	        // Buttons control
	        // Mains
	        IF (#statAvailAct3Mains = FALSE) THEN
	            #statAction.start := FALSE;
	            #statAction.stop := FALSE;
	            #statAction.end := FALSE;
	            
	        END_IF;
	        
	        // Cancel
	        IF (#statAvailActCancel = FALSE) THEN
	            #statAction.cancel := FALSE;
	            
	        END_IF;
	        
	        // Confirm
	        IF (#statAvailActConfirm = FALSE) THEN
	            #statAction.confirm := FALSE;
	            
	        END_IF;
	        
	        // Reset time
	        IF (#statAvailActResetTime = FALSE) THEN
	            #statAction.resetTime := FALSE;
	            
	        END_IF;
	        
	        // Action: Collective integer
	        "AFC_Struct_To_Word"(s := #statAction,
	                             w => #tempAction);
	        
	        #action := WORD_TO_INT(#tempAction);
	        
	    END_REGION reset availability and latching buttons
	    
	END_REGION CONTROL OPTIONS
	
	REGION WRITE OUTPUTS
	    // Outputs
	    #availAct3Mains := #statAvailAct3Mains;
	    #availActCancel := #statAvailActCancel;
	    #availActConfirm := #statAvailActConfirm;
	    #availActResetTime := #statAvailActResetTime;
	    
	END_REGION WRITE OUTPUTS
END_FUNCTION_BLOCK

FUNCTION_BLOCK "AFB_Sequencer"
TITLE = AFB_Sequencer1
{ S7_Optimized_Access := 'TRUE' }
AUTHOR : CH
FAMILY : Aktina
NAME : SEQUENCER
VERSION : 0.1
//AFB_Sequencer1
   VAR_INPUT 
      p1s : Bool;   //  TRUE: 1 pulse every 1s
      startAllow : Bool;   //  TRUE: The sequencer start condition is valid and it is allowed to start
      startCond : Bool;   //  TRUE: The options controller released the condition for the booting of the sequencer
      endCond : Bool;   //  TRUE: The state machine should end its execution immediately
      runcond : Bool;   //  TRUE: The option is running
      resetTimeOut : Bool;   //  TRUE: The time out timer should reset
      offset : Int;   //  Offset number for active step
      holdReset : DInt;   //  Preset time after the end of the sequencer to block restarting
      stepSP : Array[0..#ctMAX_STEP] of "dtStepSP";   //  Array containing the steps setpoints
      stepCond : Array[0..#ctMAX_STEP] of "dtStepCond";   //  Array containing all the steps conditions
   END_VAR

   VAR_OUTPUT 
      blocked : Bool;   //  TRUE: The sequencer is blocked from starting
      timeout : Bool;   //  TRUE: The sequencer execution has timed out
      busy : Bool;   //  TRUE: The sequencer has started and it is ongoing
      run : Bool;   //  TRUE: The sequencer operation is running
      prompt : Bool;   //  TRUE: The sequencer prompts for an operator confirmation
      error : Bool;   //  TRUE: An error was generated during execution
      noFault : Bool;   //  TRUE: The active step is running without errors
      done : Bool;   //  TRUE: The sequencer execution has finished
      terminate : Bool;   //  TRUE: The sequencer execution was terminated either by force of error
      fin : Bool;   //  TRUE: The sequencer end timer has just expired (stays high for 1 cycle)
      stepOn : Array[0..#ctMAX_STEP] of Bool;   //  TRUE: The step has just been loaded
      stepAct : Array[0..#ctMAX_STEP] of Bool;   //  TRUE: The step is active
      stepRun : Array[0..#ctMAX_STEP] of Bool;   //  TRUE: The step is running (used mostly as condition for activations)
      stepOff : Array[0..#ctMAX_STEP] of Bool;   //  TRUE: The step has just ended
      status : Word;   //  Status of the function block
      stepNr : Int;   //  Number of active step = offset + statFBState
      stateNr : Int;   //  Number of active state = statFBState
   END_VAR

   VAR RETAIN
      statStartReqOld { ExternalAccessible := 'False'; ExternalVisible := 'False'; ExternalWritable := 'False'} : Bool;
      statFBState { ExternalWritable := 'False'} : Int := #ctFB_STATE_NO_PROCESSING;   //  State in the state machine of the FB
      statStatus { ExternalWritable := 'False'} : Word := #ctSTATUS_NO_CALL;   //  Static value for output 'status'
   END_VAR
   VAR DB_SPECIFIC
      statBusy { ExternalAccessible := 'False'; ExternalVisible := 'False'; ExternalWritable := 'False'} : Bool;   //  Static value for output 'busy'
      statRun { ExternalAccessible := 'False'; ExternalVisible := 'False'; ExternalWritable := 'False'} : Bool;   //  Static value for output 'run'
      statPrompt { ExternalAccessible := 'False'; ExternalVisible := 'False'; ExternalWritable := 'False'} : Bool;   //  Static value for output 'prompt'
      statError { ExternalAccessible := 'False'; ExternalVisible := 'False'; ExternalWritable := 'False'} : Bool;   //  Static value for output 'error'
      statNoFault { ExternalAccessible := 'False'; ExternalVisible := 'False'; ExternalWritable := 'False'} : Bool;   //  Static value for output 'noFault'
      statDone { ExternalAccessible := 'False'; ExternalVisible := 'False'; ExternalWritable := 'False'} : Bool;   //  Static value for output 'done'
      statTerminate { ExternalAccessible := 'False'; ExternalVisible := 'False'; ExternalWritable := 'False'} : Bool;   //  Static value for output 'terminate'
      statFin { ExternalAccessible := 'False'; ExternalVisible := 'False'; ExternalWritable := 'False'} : Bool;   //  Static value for output 'fin'
      statExclude { S7_SetPoint := 'True'} : Bool;   //  Static value that allows the supervisor to stop the forced step updating from the current step
      statForce { S7_SetPoint := 'True'} : Bool;   //  Static value that allows the supervisor to force a new step
      statLastStep : Int;   //  Static value for the last step number
      statForceStep { S7_SetPoint := 'True'} : Int;   //  Static value for the new forced step value
   END_VAR
   VAR 
      statStepOn : Array[0..#ctMAX_STEP] of Bool;   //  Static memory area for output array "stepOn"
      statStepAct : Array[0..#ctMAX_STEP] of Bool;   //  Static memory area for output array "stepOn"
      statStepRun : Array[0..#ctMAX_STEP] of Bool;   //  Static memory area for output array "stepRun"
      statStepOff : Array[0..#ctMAX_STEP] of Bool;   //  Static memory area for output array "stepOff"
   END_VAR
   VAR RETAIN
      instTimeReset {InstructionName := 'IEC_TIMER'; LibVersion := '1.0'; S7_SetPoint := 'False'} : IEC_TIMER;   //  Instance for the timer that resets everything and prevents restarting
   END_VAR
   VAR 
      instTimeStep { S7_SetPoint := 'False'} : "AFB_TimeCount";   //  Instance for the step timer
      instTimeOut { S7_SetPoint := 'False'} : "AFB_TimeCount";   //  Instance for the timeout timer
   END_VAR

   VAR_TEMP 
      tempStartAllow : Bool;   //  Temporary status bit for the "startAllow" input
      tempStartCond : Bool;   //  Temporary status bit for the "startCond" input
      tempEndCond : Bool;   //  Temporary status bit for the "endCond" input
      tempRun : Bool;   //  Temporary status bit for the "run" input
      tempChangeStep : Bool;   //  Temporary status bit set whenever a change of step is required
      tempForceStep : Bool;   //  Temporary status bit set whenever a forcing of step is required
      tempStepSP : "dtStepSP";   //  Temporary area for the active step setpoints
      tempStepCond : "dtStepCond";   //  Temporary area for the active step conditions
      n : Int;   //  Temporary LOOP operand
   END_VAR

   VAR CONSTANT 
      ctMAX_STEP : Int := 31;   //  Max: Number steps
      ctMAX_HOPS : Int := 31;   //  Max: Hops allowed for the while loop
      ctFB_STATE_NO_PROCESSING : Int := 0;   //  FB state: No processing
      ctFB_STATE_PROCESSING_1 : Int := 1;   //  FB state: Processing 1
      ctSTATUS_NO_CALL : Word := 16#7000;   //  Status: No job being currently processed
      ctSTATUS_FIRST_CALL : Word := 16#7001;   //  Status: First call after incoming new job (rising edge 'execute')
      ctSTATUS_SUBSEQUENT_CALL : Word := 16#7002;   //  Status: Subsequent call during active processing without further details
      ctSTATUS_EXECUTION_TERMINATED : Word := 16#7008;   //  Status: Execution finished without errors
      ctSTATUS_EXECUTION_FINISHED : Word := 16#700F;   //  Status: Execution finished without errors
      ctERR_UNDEFINED_STATE : Word := 16#8000;   //  Error: Due to an undefined state in state machine
      ctERR_IN_BLOCK_OPERATION : Word := 16#8001;   //  Error: Wrong operation of the function block
      ctERR_PARAMETRIZATION : Word := 16#8002;   //  Error: During parameterization
   END_VAR


BEGIN
	REGION BLOCK HEADER
	     //===============================================================================
	     // CH / (c)Copyright (2021)
	     //-------------------------------------------------------------------------------
	     // Title:             (Sequencer control block type 1)
	     // Comment/Function:  (Control step execution of a sequencer by providing only key conditions and setpoints)
	     // Library/Family:    (Aktina/Tools/Sequencer)
	     // Author:            (CH)
	     // Tested with:       (V16)
	     // Engineering:       (TIA Step7 Professional V16)
	     // Restrictions:      ()
	     // Requirements:      (S7-15xx/12xx CPUs)
	     // Notes:             (See block notes)
	     //-------------------------------------------------------------------------------
	     // Change log table:
	     // Version  | Date       | Dev in charge          | Changes
	     //----------|------------|------------------------|------------------------------
	     // 01.00.00 | 2021-08-22 | (CH)                   | First released version
	     // 01.00.01 | 2022-01-13 | (CH)                   | "No timeout" allowed - busy hangon corrected
	     // 01.00.02 | 2023-05-18 | (CH)                   | "RESET(instResetTimer) - removed to allow timer to run
	     //===============================================================================
	END_REGION
	
	REGION BLOCK NOTES
	     //===============================================================================
	     // 1: The number of steps participating is configured by the #ctMAX_STEP
	     //-------------------------------------------------------------------------------
	     // 2: The idle or exit step is always 0 so the number of steps remaining
	     // for the rest of the program is steps = #ctMAX_Step - 1
	     //-------------------------------------------------------------------------------
	     // 3: The block supports zero cycles for step change even if there are 
	     // multiple hops.
	     //-------------------------------------------------------------------------------
	     // 4: The maximum allowed number of hops is the ctMAX_HOPS to avoid an endless
	     // loop. After that alarm is generated.
	     //===============================================================================
	END_REGION
	
	REGION GENERIC PRE-INSTRUCTIONS
	     //  Init temporary area
	     #tempStartAllow := (#startAllow = TRUE) AND (#instTimeReset.Q = FALSE) AND (#statDone = FALSE) AND (#statTerminate = FALSE);
	     #tempStartCond := #startCond;
	     #tempEndCond := #endCond;
	     #tempRun := #runcond;
	     #tempChangeStep := FALSE;
	     #tempForceStep := FALSE;
	     #tempStepSP := #stepSP[0];
	     #tempStepCond := #stepCond[0];
	     #n := 0;
	     
	     // Reset static step memory with every cycle to avoid forced states loaded by a programmer
	     FOR #n := 0 TO #ctMAX_STEP DO
	          #statStepOn[#n] := FALSE;
	          #statStepAct[#n] := FALSE;
	          #statStepRun[#n] := FALSE;
	          #statStepOff[#n] := FALSE;
	     END_FOR;
	     
	END_REGION GENERIC PRE-INSTRUCTIONS
	
	REGION TRIGGERING
	     IF (#tempStartCond = TRUE) AND (#statStartReqOld = FALSE) // Check if FB is triggered
	          AND (#tempStartAllow = TRUE)
	          AND (#tempEndCond = FALSE)
	          AND (#instTimeReset.Q = FALSE)
	          AND (#stepSP[0].next > 0)
	          AND (#statBusy = FALSE)
	          AND (#statDone = FALSE)
	     THEN // First call; initialize FB stat 
	          // TODO: Initialize functionality: reset of variables, diagnostics, etc.
	          #statBusy := TRUE;
	          #statStepOff[0] := TRUE;
	          #statStepAct[0] := FALSE;
	          #statStatus := #ctSTATUS_FIRST_CALL;
	          
	          // TODO: Initialize functionality: start state machine.
	          #statFBState := #stepSP[0].next;
	          
	          // TODO: Initialize functionality: call subsidiary FBs with FALSE
	          "AFC_RESET_TimeCount"(#instTimeStep);
	          "AFC_RESET_TimeCount"(#instTimeOut);
	          RESET_TIMER(#instTimeReset);
	          
	     ELSIF (#statStatus = #ctSTATUS_FIRST_CALL) THEN
	          #statStatus := #ctSTATUS_SUBSEQUENT_CALL;
	     END_IF;
	     
	     // Edge detection 'startReq' input
	     #statStartReqOld := #tempStartCond;
	END_REGION TRIGGERING
	
	REGION END WHEN IDLE
	     IF (#statStatus = #ctSTATUS_NO_CALL) THEN // Nothing to do -> End here to reduce "system load"
	          // Static memory
	          #statDone := FALSE;
	          #statTerminate := FALSE;
	          #statBusy := FALSE;
	          #statRun := FALSE;
	          #statNoFault := TRUE;
	          #statError := FALSE;
	          #statPrompt := FALSE;
	          #statExclude := FALSE;
	          #statForce := FALSE;
	          #statFin := FALSE;
	          #statLastStep := #statFBState;
	          #statForceStep := #statFBState;
	          #statStepAct[0] := TRUE;
	          
	          // if ENO mechanism is not used / not wanted replace the following line by --> ENO := TRUE;
	          // ENO := NOT #statError;
	          ENO := TRUE;
	          
	          // Outputs
	          #blocked := (#startAllow = FALSE);
	          #timeout := FALSE;
	          #done := #statDone;
	          #terminate := #statTerminate;
	          #busy := #statBusy;
	          #run := #statRun;
	          #noFault := #statNoFault;
	          #error := #statError;
	          #prompt := #statPrompt;
	          #fin := #statFin;
	          #stepOn := #statStepOn;
	          #stepAct := #statStepAct;
	          #stepRun := #statStepRun;
	          #stepOff := #statStepOff;
	          #status := #statStatus;
	          #stepNr := #statFBState + #offset;
	          #stateNr := #statFBState;
	          
	          RETURN;
	          
	     END_IF;
	     
	END_REGION END WHEN IDLE
	
	REGION STATE_MACHINE
	     
	     CASE #statFBState OF // State machine of FB
	               
	          #ctFB_STATE_NO_PROCESSING:
	               REGION no processing
	                    // No processing active (Note: this state must always be present and left empty)
	                    ;
	               END_REGION no processing
	               
	          #ctFB_STATE_PROCESSING_1..#ctMAX_STEP: // Processing active
	               REGION processing n-step
	                    // Processing active n=#statFBState case is processed
	                    // The goal is to run the step with the minimum system load
	                    // If a step change is required it is done in the same programming cycle 
	                    
	                    // The step conditions are evaluated in a WHILE loop and the loop
	                    // is interrupted whenever a valid step is loaded or the maximum 
	                    // allowed hops are counted
	                    
	                    #n := 0;
	                    WHILE (#n <= #ctMAX_HOPS) DO
	                         // Increase operand by 1 with each loop
	                         #n := #n + 1;
	                         
	                         // Scan the state of the machine for the end condition
	                         IF (#statFBState = 0)
	                         THEN
	                              #statStatus := #ctSTATUS_EXECUTION_FINISHED;
	                              
	                         ELSIF (#tempEndCond = TRUE) OR (#statBusy = FALSE)
	                         THEN
	                              #statStatus := #ctSTATUS_EXECUTION_TERMINATED;
	                              
	                         ELSIF (#statFBState < 0) OR (#statFBState > #ctMAX_STEP)
	                              OR (#ctMAX_STEP < 2)
	                         THEN
	                              #statStatus := #ctERR_IN_BLOCK_OPERATION;
	                              
	                         ELSIF (#n >= #ctMAX_HOPS)
	                         THEN
	                              #statStatus := #ctERR_PARAMETRIZATION;
	                              
	                         END_IF;
	                         
	                         // Exit loop if a status of aborting is detected
	                         IF (#statStatus >= #ctSTATUS_EXECUTION_TERMINATED)
	                         THEN
	                              
	                              EXIT; // exit loop immediately
	                              
	                         END_IF;
	                         
	                         // Move active step data to temporary area for the eaase of use
	                         #tempStepSP := #stepSP[#statFBState];
	                         #tempStepCond := #stepCond[#statFBState];
	                         
	                         // Load correct arguments to the timers
	                         #instTimeStep.preset := #tempStepSP.timeStep;
	                         #instTimeOut.preset := #tempStepSP.timeOut;
	                         
	                         // Condition to change a step
	                         #tempChangeStep := (#tempRun = TRUE) AND (
	                         (#tempStepSP.type = 0) AND (#instTimeStep.done = TRUE) OR
	                         (#tempStepSP.type = 1) AND (#tempStepCond.proceed = TRUE) OR
	                         (#tempStepSP.type = 2) AND (#instTimeStep.done = TRUE) AND (#tempStepCond.proceed = TRUE)
	                         );
	                         
	                         // Condition to force a new step
	                         #tempForceStep := (#statExclude = TRUE)
	                         AND (#statForceStep <= #ctMAX_STEP) AND (#statForceStep > 0)
	                         AND (#statForce = TRUE);
	                         
	                         // Scan the state of the machine for a change step condition
	                         IF (#tempChangeStep = TRUE)
	                         THEN
	                              #statStepAct[#statFBState] := FALSE;
	                              #statStepOff[#statFBState] := TRUE;
	                              #statNoFault := TRUE;
	                              #statPrompt := FALSE;
	                              #statLastStep := #statFBState;
	                              #statFBState := #tempStepSP.next;
	                              #statStepOn[#statFBState] := TRUE;
	                              
	                              "AFC_RESET_TimeCount"(#instTimeStep);
	                              "AFC_RESET_TimeCount"(#instTimeOut);
	                              
	                              CONTINUE; // Rerun loop to check the new step's conditions in case an immediate change is requested.
	                              
	                         ELSIF (#tempForceStep = TRUE)
	                         THEN
	                              #statStepAct[#statFBState] := FALSE;
	                              #statStepRun[#statFBState] := FALSE;
	                              #statStepOff[#statFBState] := TRUE;
	                              #statNoFault := TRUE;
	                              #statPrompt := FALSE;
	                              #statLastStep := #statFBState;
	                              #statFBState := #statForceStep;
	                              #statStepOn[#statFBState] := TRUE;
	                              
	                              #statExclude := FALSE;
	                              #statForce := FALSE;
	                              
	                              "AFC_RESET_TimeCount"(#instTimeStep);
	                              "AFC_RESET_TimeCount"(#instTimeOut);
	                              
	                              CONTINUE; // Rerun loop to check the new step's conditions in case an immediate change is requested.
	                              
	                         END_IF;
	                         
	                         // If the loop reaches this point then the step=#statFBState is active
	                         EXIT;
	                         
	                    END_WHILE;
	                    
	                    #statStepAct[#statFBState] := TRUE;
	                    #statStepRun[#statFBState] := #tempRun;
	                    
	                    #instTimeStep.trigger := #tempStepCond.count;
	                    #instTimeStep.reset := #tempStepCond.reset;
	                    
	                    #instTimeOut.trigger := TRUE;
	                    
	                    IF (#statExclude = FALSE) THEN
	                         #statForceStep := #statFBState;
	                    END_IF;
	                    
	                    #statNoFault := #tempStepCond.nofault;
	                    #statPrompt := #tempStepCond.prompt;
	                    #statRun := #tempRun;
	                    
	               END_REGION processing n-step      
	               
	          ELSE // Undefined state in state machine reached
	               REGION undefined state
	                    #statStatus := #ctERR_UNDEFINED_STATE;
	                    
	               END_REGION undefined state
	     END_CASE;
	END_REGION STATE_MACHINE
	
	REGION OUTPUTS
	     // Write outputs
	     IF (#statStatus = #ctSTATUS_EXECUTION_FINISHED) AND (#statDone = FALSE) THEN // Execution finished without errors
	          REGION execution finished
	               #statDone := TRUE;
	               #statTerminate := FALSE;
	               #statBusy := FALSE;
	               #statError := FALSE;
	               #statExclude := FALSE;
	               #statForce := FALSE;
	               #statNoFault := TRUE;
	               #statPrompt := FALSE;
	               #statStepOn[0] := TRUE;
	               #statStepAct[0] := TRUE;
	               
	               // reset step timers
	               "AFC_RESET_TimeCount"(#instTimeStep);
	               "AFC_RESET_TimeCount"(#instTimeOut);
	               
	               // reset state machine
	               #statFBState := #ctFB_STATE_NO_PROCESSING;
	               
	          END_REGION execution finished
	          
	     ELSIF (#statStatus = #ctSTATUS_EXECUTION_TERMINATED) AND (#statTerminate = FALSE) THEN // Execution forced to stop
	          REGION execution terminated
	               #statDone := FALSE;
	               #statTerminate := TRUE;
	               #statBusy := FALSE;
	               #statError := FALSE;
	               #statExclude := FALSE;
	               #statForce := FALSE;
	               #statNoFault := TRUE;
	               #statPrompt := FALSE;
	               #statStepOn[0] := TRUE;
	               #statStepAct[0] := TRUE;
	               
	               // reset step timers
	               "AFC_RESET_TimeCount"(#instTimeStep);
	               "AFC_RESET_TimeCount"(#instTimeOut);
	               
	               // reset state machine
	               #statFBState := #ctFB_STATE_NO_PROCESSING;
	               
	          END_REGION execution terminated
	          
	     ELSIF (#statStatus.%X15 = TRUE) AND (#statError = FALSE) THEN // Error occurred (#statStatus is 16#8000 to 16#FFFF)
	          REGION error occured
	               #statDone := FALSE;
	               #statTerminate := TRUE;
	               #statBusy := FALSE;
	               #statError := TRUE;
	               #statExclude := FALSE;
	               #statForce := FALSE;
	               #statNoFault := TRUE;
	               #statPrompt := FALSE;
	               #statStepOn[0] := TRUE;
	               #statStepAct[0] := TRUE;
	               
	               // reset step timers
	               "AFC_RESET_TimeCount"(#instTimeStep);
	               "AFC_RESET_TimeCount"(#instTimeOut);
	               
	               // reset state machine
	               #statFBState := #ctFB_STATE_NO_PROCESSING;
	               
	          END_REGION error occured
	          
	     ELSIF (#instTimeReset.Q = FALSE) AND ((#statDone = TRUE) OR (#statTerminate = TRUE)) THEN // Reset outputs //    AND (#statBusy = FALSE)  // CH: 20230518 - Changed to allow total reset when timer is running
	          REGION execute total reset
	               #statDone := FALSE;
	               #statTerminate := FALSE;
	               #statBusy := FALSE;
	               #statError := FALSE;
	               #statExclude := FALSE;
	               #statForce := FALSE;
	               #statFin := TRUE;
	               // reset status
	               #statStatus := #ctSTATUS_NO_CALL;
	               
	               // reset state machine
	               #statFBState := #ctFB_STATE_NO_PROCESSING;
	               #statLastStep := #statFBState;
	               
	               // TODO: Reset application specific outputs
	               "AFC_RESET_TimeCount"(#instTimeStep);
	               "AFC_RESET_TimeCount"(#instTimeOut);
	               RESET_TIMER(#instTimeReset);
	               
	          END_REGION execute total reset
	     END_IF;
	     
	     REGION timers
	          // Call instances
	          #instTimeStep(p1s := #p1s);
	          
	          #instTimeOut(p1s := #p1s,
	                       reset := #resetTimeOut);
	          
	          // **Added to allow "no timeout" setup
	          IF (#instTimeOut.statPresetSec = 0)
	          THEN
	               "AFC_RESET_TimeCount"(#instTimeOut);
	          END_IF;
	          
	          #instTimeReset.TOF(IN := (#statBusy = TRUE),
	                             PT := DINT_TO_TIME(#holdReset));
	          
	     END_REGION timers
	     
	     REGION write static values to outputs
	          // if ENO mechanism is not used / not wanted replace the following line by --> ENO := TRUE;
	          // ENO := NOT #statError;
	          ENO := TRUE;
	          // TODO: Write application specific static values to outputs
	          #blocked := (#instTimeReset.Q = TRUE) AND (#statBusy = FALSE);
	          #timeout := (#instTimeOut.done = TRUE) AND (#statBusy = TRUE);
	          #done := #statDone;
	          #terminate := #statTerminate;
	          #busy := #statBusy;
	          #run := #statRun;
	          #noFault := #statNoFault;
	          #error := #statError;
	          #prompt := #statPrompt;
	          #fin := #statFin;
	          #stepOn := #statStepOn;
	          #stepAct := #statStepAct;
	          #stepRun := #statStepRun;
	          #stepOff := #statStepOff;
	          #status := #statStatus;
	          #stepNr := #statFBState + #offset;
	          #stateNr := #statFBState;
	          
	     END_REGION write static values TO outputs
	     
	END_REGION OUTPUTS
END_FUNCTION_BLOCK

FUNCTION_BLOCK "AFB_TimeCount"
TITLE = AFB_HoursCounter
{ S7_Optimized_Access := 'TRUE' }
AUTHOR : CH
FAMILY : Aktina
NAME : 'TIME'
VERSION : 0.1
//AFB_HoursCounter
   VAR_INPUT 
      trigger { ExternalAccessible := 'False'; ExternalVisible := 'False'; ExternalWritable := 'False'} : Bool;   //  TRUE: Run timer
      reset { ExternalAccessible := 'False'; ExternalVisible := 'False'; ExternalWritable := 'False'} : Bool;   //  TRUE: Reset timer
      p1s { ExternalAccessible := 'False'; ExternalVisible := 'False'; ExternalWritable := 'False'} : Bool;   //  TRUE: 1 second pulse
      preset : "dtTimerArguments";   //  Preset timer arguments
   END_VAR

   VAR_OUTPUT 
      done : Bool;   //  TRUE: Preset time elapsed
      remain : "dtTimerArguments";   //  Remaining timer arguments
   END_VAR

   VAR 
      statPresetSec : UDInt;   //  Static value for preset time
   END_VAR
   VAR RETAIN
      statSec : UDInt;   //  Static value for seconds counted
      statRem : Struct   //  Static value for minutes remaining
         sec : UDInt;   //  seconds
         min : UDInt;   //  minutes
         hour : UDInt;   //  hours
      END_STRUCT;
   END_VAR

   VAR_TEMP 
      tempTrigger : Bool;   //  Temporary value for input 'trigger'
      tempReset : Bool;   //  Temporary value for input 'reset'
   END_VAR


BEGIN
	REGION BLOCK HEADER
	     //===============================================================================
	     // CH / (c)Copyright (2021)
	     //-------------------------------------------------------------------------------
	     // Title:             (Hours counter)
	     // Comment/Function:  (Hours counter)
	     // Library/Family:    (Aktina/Tools/Time)
	     // Author:            (CH)
	     // Tested with:       (V16)
	     // Engineering:       (TIA Step7 Professional V16)
	     // Restrictions:      ()
	     // Requirements:      (S7 CPUs)
	     // Notes:             ()
	     //-------------------------------------------------------------------------------
	     // Change log table:
	     // Version  | Date       | Dev in charge          | Changes
	     //----------|------------|------------------------|------------------------------
	     // 01.00.00 | 2021-03-13 | (CH)                   | First released version
	     //===============================================================================
	END_REGION
	
	REGION GENERIC PRE-INSTRUCTIONS
	     // Work with temporary value / create process image
	     #tempReset := #reset;
	     #tempTrigger := (#tempReset = FALSE) AND (#trigger = TRUE) AND (#p1s = TRUE);
	END_REGION GENERIC PRE-INSTRUCTIONS
	
	REGION END WHEN RESET
	     IF (#tempReset = TRUE)
	     THEN // Nothing to do -> End here to reduce "system load"
	          #statSec := 0;
	          #statPresetSec := 0;
	          #statRem.sec := 0;
	          #statRem.min := 0;
	          #statRem.hour := 0;
	          #remain.sec := 0;
	          #remain.min := 0;
	          #remain.hour := 0;
	          #done := FALSE;
	          RETURN;
	     END_IF;
	     
	END_REGION END WHEN RESET
	
	REGION TIMER
	     #statPresetSec := (UINT_TO_UDINT(#preset.hour) * 3600) + (USINT_TO_UDINT(#preset.min) * 60) + USINT_TO_UDINT(#preset.sec);
	     
	     IF (#tempTrigger = TRUE) AND (#statSec < #statPresetSec)
	     THEN
	          #statSec := #statSec + 1;
	     END_IF;
	END_REGION TIMER
	
	REGION OUTPUT
	     #done := ((#trigger = TRUE) AND (#statPresetSec = 0)) OR ((#statSec >= #statPresetSec) AND (#statPresetSec > 0));
	     
	     #statRem.sec := #statPresetSec - #statSec;
	     
	     #statRem.hour := #statRem.sec / 3600;
	     #statRem.min := (#statRem.sec / 60) - (#statRem.hour * 60);
	     
	     #remain.sec := UDINT_TO_USINT(#statRem.sec - (#statRem.min * 60) - (#statRem.hour * 3600));
	     #remain.min := UDINT_TO_USINT(#statRem.min);
	     #remain.hour := UDINT_TO_USINT(#statRem.hour);
	END_REGION OUTPUT
	
END_FUNCTION_BLOCK

FUNCTION "AFC_RESET_TimeCount" : Void
TITLE = AFC_RESET_HoursCounter
{ S7_Optimized_Access := 'TRUE' }
AUTHOR : CH
FAMILY : Aktina
NAME : 'TIME'
VERSION : 0.1
//AFC_RESET_HoursCounter
   VAR_IN_OUT 
      hoursCounter : "AFB_TimeCount";   //  Hours counter to be reset
   END_VAR


BEGIN
	// Reset timer totally
	
	#hoursCounter.trigger := FALSE;
	#hoursCounter.reset := TRUE;
	
	#hoursCounter.preset.sec := 0;
	#hoursCounter.preset.min := 0;
	#hoursCounter.preset.hour := 0;
	
	#hoursCounter();
	
	#hoursCounter.reset := FALSE;
	
END_FUNCTION

FUNCTION "getStepState" : Void
{ S7_Optimized_Access := 'TRUE' }
VERSION : 0.1
   VAR_INPUT 
      index : Int;
      step : Struct
         ON : Array[0..31] of Bool;
         OFF : Array[0..31] of Bool;
         ACT : Array[0..31] of Bool;
         RUN : Array[0..31] of Bool;
      END_STRUCT;
   END_VAR

   VAR_OUTPUT 
      run : Bool;
      act : Bool;
      off : Bool;
      on : Bool;
   END_VAR


BEGIN
	#run := #step.RUN[#index];
	#act := #step.ACT[#index];
	#on := #step.ON[#index];
	#off := #step.OFF[#index];
END_FUNCTION

FUNCTION_BLOCK "libCpu_SystemInfo"
{ S7_Optimized_Access := 'TRUE' }
AUTHOR : CH
FAMILY : Aktina
NAME : Lib_System
VERSION : 1.1
   VAR_INPUT 
      init { ExternalAccessible := 'False'; ExternalVisible := 'False'; ExternalWritable := 'False'} : Bool;   //  TRUE: First cycle
      clockByte { ExternalWritable := 'False'} : Byte;   //  Clock byte provided by the CPU
   END_VAR

   VAR_OUTPUT 
      timeByte { ExternalWritable := 'False'} : Byte;   //  Time byte resulting as PPD of 'clockByte'
      localTime {InstructionName := 'DTL'; LibVersion := '1.0'} : DTL;   //  Local CPU time
   END_VAR

   VAR RETAIN
      statLocalTime {InstructionName := 'DTL'; LibVersion := '1.0'; ExternalWritable := 'False'} : DTL;
      statClockByteOld { ExternalWritable := 'False'} : Byte;
   END_VAR
   VAR 
      statTimeByte { ExternalWritable := 'False'} : Byte;
   END_VAR

   VAR_TEMP 
      tempClockByte : Byte;
      tempLocalTimeRet : Int;
   END_VAR


BEGIN
	//===============================================================================
	// Aktinaplan Ltd / (c)Copyright (2023)
	//-------------------------------------------------------------------------------
	// Title:            (System bits)
	// Comment/Function: ()
	// Library/Family:   (Aktina/Tools/System)
	// Author:           (CH)
	// Tested with:      (S7 1513)
	// Engineering:      TIA Portal (v15.1)
	// Restrictions:     ()
	// Requirements:     (S7)
	//-------------------------------------------------------------------------------
	// Change log table:
	// Version  | Date       | Expert in charge       | Changes applied
	//----------|------------|------------------------|------------------------------
	// 01.00.00 | 2023-01-08 | CH                     | First released version
	// 01.00.01 | 2023-07-28 | CH                     | Added local time
	//===============================================================================
	
	REGION Initialization
	     
	     IF (#init = TRUE) THEN
	          // initialize memory
	          #statClockByteOld := 16#0;
	          #statTimeByte := 16#0;
	          #timeByte := 16#0;
	          // and exit block
	          RETURN;
	     END_IF;
	     
	END_REGION
	
	REGION Local PI
	     // Create process image
	     #tempClockByte := #clockByte;
	     
	END_REGION
	
	REGION Instructions
	     // System instruction (write under here the instructions)
	     
	     REGION Cpu time byte    
	          // Create time byte based on ppd detection of Cpu frequency bits
	          #statTimeByte := #tempClockByte XOR #statClockByteOld AND #tempClockByte;
	          // Edge detection
	          #statClockByteOld := #clockByte;
	          
	     END_REGION
	     
	     REGION CPU local time
	          // Read local time instruction
	          #tempLocalTimeRet := RD_LOC_T(#statLocalTime);
	          
	     END_REGION
	     
	END_REGION
	
	REGION Outputs
	     // Block outputs
	     #timeByte := #statTimeByte;
	     #localTime := #statLocalTime;
	     
	END_REGION ;
	
END_FUNCTION_BLOCK

FUNCTION "Indications" : Void
{ S7_Optimized_Access := 'TRUE' }
VERSION : 0.1
   VAR_TEMP 
      tempLastTT : Real;   //  Temporary value for the last temperature transmitter output
   END_VAR


BEGIN
	REGION Cabinet ( number of cabinet )
	
	    // Indication: Beacon operating GREEN color
	    
	    
	    // Indication: Beacon "Fault" RED color
	
	    
	    // Indication: Beacon Siren
	    
	    
	    // Indication: Led blue of reset button
	    
	    
	    // Indication: Reset
	     
	        
	 END_REGION
	
	 
	
END_FUNCTION

FUNCTION "quickSetup" : Void
{ S7_Optimized_Access := 'TRUE' }
VERSION : 0.1
   VAR_IN_OUT 
      setup : "modTypes";   //  TRUE: Quick setup of the selected type
   END_VAR

   VAR_TEMP 
      i : DInt;   //  Temporary indexer
   END_VAR


BEGIN
	
	REGION PUT / GET
	    // Statement section REGION
	    "GET_DB"(REQ:="p100ms",
	             ID:=W#16#100,
	             ADDR_1:=P#I512.0 DWORD 8,
	             RD_1:=P#M512.0 DWORD 8);
	
	END_REGION
	
	REGION sim
	    FOR #i := 0 TO "M_MTRDIR" DO
	        "MODULES_CTRL".MTRDIR[#i].status := TRUE;
	        // "MOD".MTRDIR[#i].i.sim.fb := FALSE;
	        // "MOD".MTRDIR[#i].i.sim.ctrl := FALSE;
	        // "MODULES_CTRL".MTRDIR[#i].sim.simFb := TRUE;
	        // "MODULES_CTRL".MTRDIR[#i].sim.simCtrl := TRUE;
	        
	        // "MOD".MTRDIR[#i].i.faults.ftr.setup.spon := 125;
	    END_FOR;
	    
	    FOR #i := 0 TO "M_MTR" DO
	        "MODULES_CTRL".MTR[#i].status := TRUE;
	        // "MOD".MTR[#i].i.sim.fb := FALSE;
	        // "MOD".MTR[#i].i.sim.ctrl := FALSE;
	        //"MODULES_CTRL".MTR[#i].sim.simFb := TRUE;
	        //"MODULES_CTRL".MTR[#i].sim.simCtrl := TRUE;
	        
	        //"MOD".MTR[#i].i.delay.in.spon := 0.5;
	    END_FOR;
	    
	    FOR #i := 0 TO "M_AIN" DO
	        "MODULES_CTRL".AIN[#i].status := TRUE;
	    END_FOR;
	    
	    FOR #i := 0 TO "M_DIN" DO
	        "MODULES_CTRL".DIN[#i].status := TRUE;
	    END_FOR;
	    
	    FOR #i := 0 TO "M_VLV" DO
	        "MODULES_CTRL".VLV[#i].status := TRUE;
	        //"MOD".VLV[#i].i.delaymain.in.spoff := 0.5;
	        // "MOD".VLV[#i].i.sim.main := TRUE;
	        // "MOD".VLV[#i].i.sim.deact := TRUE;
	    END_FOR;
	    
	    
	END_REGION
	
	
	REGION modules
	    REGION Control valves
	        
	        // IF #setup.cvlv = TRUE THEN // Setup
	        
	        //      FOR #i := 0 TO "M_CVLV" DO
	        //           "MOD".CVLV[#i].i.pid.H := 100.0;
	        //           "MOD".CVLV[#i].i.pid.mode := FALSE;
	        //           "MOD".CVLV[#i].i.unscale.inlow := 0.0;
	        //           "MOD".CVLV[#i].i.unscale.inhigh := 100.0;
	        //           "MOD".CVLV[#i].i.unscale.outlow := 4000.0;
	        //           "MOD".CVLV[#i].i.unscale.outhigh := 20000.0;
	        //      END_FOR;
	        
	        //      #setup.cvlv := FALSE; // Reset
	        
	        // END_IF;
	        
	    END_REGION Control valves     
	    
	    REGION Motors PID
	        
	        IF #setup.mtr = TRUE THEN // Setup
	            
	            FOR #i := 0 TO "M_MTR" DO
	                "MOD".MTR[#i].i.cmd.auto := TRUE;
	                "MOD".MTR[#i].i.faults.ftr.setup."en" := FALSE;
	                "MOD".MTR[#i].i.faults.ftr.setup.spon := 2.0;
	                "MOD".MTR[#i].i.faults.fts.setup."en" := FALSE;
	                "MOD".MTR[#i].i.faults.fts.setup.spon := 6.0;
	                "MOD".MTR[#i].i.faults.mcb.setup."en" := FALSE;
	                "MOD".MTR[#i].i.faults.mcb.setup.spon := 2.0;
	                "MOD".MTR[#i].i.faults.ctrl.setup."en" := FALSE;
	                "MOD".MTR[#i].i.faults.ctrl.setup.spon := 2.0;
	                "MOD".MTR[#i].i.faults.vfd.setup."en" := FALSE;
	                "MOD".MTR[#i].i.faults.vfd.setup.spon := 5.0;
	                "MOD".MTR[#i].i.unscale.inhigh := 100.0;
	                "MOD".MTR[#i].i.unscale.outhigh := 100.0;
	                "MOD".MTR[#i].i.pid.L := 10.0;
	                "MOD".MTR[#i].i.pid.H := 100.0;
	                "MOD".MTR[#i].i.pid.OP := 50.0;
	                "MOD".MTR[#i].i.pid.P := 0.5;
	                "MOD".MTR[#i].i.pid.I := 8000;
	                "MOD".MTR[#i].i.pid.outunit := WSTRING#'%';
	                
	                "MOD".MTR[#i].i.pid.mode := TRUE;
	                
	            END_FOR;
	            
	            #setup.mtr := FALSE; // Reset
	            
	        END_IF;
	        
	    END_REGION Motors PID
	    
	    REGION Valves
	        
	        IF #setup.vlv = TRUE THEN
	            
	            FOR #i := 0 TO "M_VLV" DO // Setup
	                "MOD".VLV[#i].i.faults.ftamain.setup."en" := TRUE;
	                "MOD".VLV[#i].i.faults.ftamain.setup.spon := 6.0;
	                "MOD".VLV[#i].i.faults.ftd.setup."en" := TRUE;
	                "MOD".VLV[#i].i.faults.ftd.setup.spon := 6.0;
	                
	            END_FOR;
	            
	            #setup.vlv := FALSE; // Reset
	            
	        END_IF;
	        
	    END_REGION Valves
	    
	    REGION Analog sensors
	        
	        IF #setup.ain = TRUE THEN
	            FOR #i := 0 TO 5 DO
	                "MOD".AIN[#i].i.chn.type := 2;
	                "MOD".AIN[#i].i.scale.factor := 0.01;
	                "MOD".AIN[#i].i.unit := WSTRING#'mbar';
	                
	            END_FOR;
	            
	            FOR #i := 6 TO 11 DO
	                "MOD".AIN[#i].i.chn.type := 2;
	                "MOD".AIN[#i].i.scale.factor := 0.1;
	                "MOD".AIN[#i].i.unit := WSTRING#'°C';
	                
	            END_FOR;
	            
	        END_IF;
	        
	        // Reset
	        #setup.ain := FALSE;
	        
	    END_REGION Analog sensors
	    
	    #i := 0;
	END_REGION
	
END_FUNCTION

FUNCTION_BLOCK "AFB_HoursCounter"
TITLE = AFB_HoursCounter
{ S7_Optimized_Access := 'TRUE' }
AUTHOR : CH
FAMILY : Aktina
NAME : 'TIME'
VERSION : 0.1
//AFB_HoursCounter
   VAR_INPUT 
      trigger { ExternalAccessible := 'False'; ExternalVisible := 'False'; ExternalWritable := 'False'} : Bool;   //  TRUE: Run timer
      reset { ExternalAccessible := 'False'; ExternalVisible := 'False'; ExternalWritable := 'False'} : Bool;   //  TRUE: Reset timer
      p1s { ExternalAccessible := 'False'; ExternalVisible := 'False'; ExternalWritable := 'False'} : Bool;   //  TRUE: 1 second pulse
      preset : "dtTimerArguments";   //  Preset timer arguments
   END_VAR

   VAR_OUTPUT 
      done : Bool;   //  TRUE: Preset time elapsed
      remain : "dtTimerArguments";   //  Remaining timer arguments
   END_VAR

   VAR 
      statPresetSec : UDInt;   //  Static value for preset time
   END_VAR
   VAR RETAIN
      statSec : UDInt;   //  Static value for seconds counted
      statRem : Struct   //  Static value for minutes remaining
         sec : UDInt;   //  seconds
         min : UDInt;   //  minutes
         hour : UDInt;   //  hours
      END_STRUCT;
   END_VAR

   VAR_TEMP 
      tempTrigger : Bool;   //  Temporary value for input 'trigger'
      tempReset : Bool;   //  Temporary value for input 'reset'
   END_VAR


BEGIN
	REGION BLOCK HEADER
	    //===============================================================================
	    // CH / (c)Copyright (2021)
	    //-------------------------------------------------------------------------------
	    // Title:             (Hours counter)
	    // Comment/Function:  (Hours counter)
	    // Library/Family:    (Aktina/Tools/Time)
	    // Author:            (CH)
	    // Tested with:       (V16)
	    // Engineering:       (TIA Step7 Professional V16)
	    // Restrictions:      ()
	    // Requirements:      (S7 CPUs)
	    // Notes:             ()
	    //-------------------------------------------------------------------------------
	    // Change log table:
	    // Version  | Date       | Dev in charge          | Changes
	    //----------|------------|------------------------|------------------------------
	    // 01.00.00 | 2021-03-13 | (CH)                   | First released version
	    //===============================================================================
	END_REGION
	
	REGION GENERIC PRE-INSTRUCTIONS
	    // Work with temporary value / create process image
	    #tempReset := #reset;
	    #tempTrigger := (#tempReset = FALSE) AND (#trigger = TRUE) AND (#p1s = TRUE);
	END_REGION GENERIC PRE-INSTRUCTIONS
	
	REGION END WHEN RESET
	    IF (#tempReset = TRUE)
	    THEN // Nothing to do -> End here to reduce "system load"
	        #statSec := 0;
	        #statPresetSec := 0;
	        #statRem.sec := 0;
	        #statRem.min := 0;
	        #statRem.hour := 0;
	        #remain.sec := 0;
	        #remain.min := 0;
	        #remain.hour := 0;
	        #done := FALSE;
	        RETURN;
	    END_IF;
	    
	END_REGION END WHEN RESET
	
	REGION TIMER
	    #statPresetSec := (UINT_TO_UDINT(#preset.hour) * 3600) + (USINT_TO_UDINT(#preset.min) * 60) + USINT_TO_UDINT(#preset.sec);
	    
	    IF (#tempTrigger = TRUE) AND (#statSec < #statPresetSec)
	    THEN
	        #statSec := #statSec + 1;
	    END_IF;
	END_REGION TIMER
	
	REGION OUTPUT
	    #done := ((#trigger = TRUE) AND (#statPresetSec = 0)) OR ((#statSec >= #statPresetSec) AND (#statPresetSec > 0));
	    
	    #statRem.sec := #statPresetSec - #statSec;
	    
	    #statRem.hour := #statRem.sec / 3600;
	    #statRem.min := (#statRem.sec / 60) - (#statRem.hour * 60);
	    
	    #remain.sec := UDINT_TO_USINT(#statRem.sec - (#statRem.min * 60) - (#statRem.hour * 3600));
	    #remain.min := UDINT_TO_USINT(#statRem.min);
	    #remain.hour := UDINT_TO_USINT(#statRem.hour);
	END_REGION OUTPUT
	
END_FUNCTION_BLOCK

FUNCTION "AFC_RESET_HoursCounter" : Void
TITLE = AFC_RESET_HoursCounter
{ S7_Optimized_Access := 'TRUE' }
AUTHOR : CH
FAMILY : Aktina
NAME : 'TIME'
VERSION : 0.1
//AFC_RESET_HoursCounter
   VAR_IN_OUT 
      hoursCounter : "AFB_HoursCounter";   //  Hours counter to be reset
   END_VAR


BEGIN
	// Reset timer totally
	
	#hoursCounter.trigger := FALSE;
	#hoursCounter.reset := TRUE;
	
	#hoursCounter.preset.sec := 0;
	#hoursCounter.preset.min := 0;
	#hoursCounter.preset.hour := 0;
	
	#hoursCounter();
	
	#hoursCounter.reset := FALSE;
	
END_FUNCTION

FUNCTION_BLOCK "AFB_MODULES"
{ S7_Optimized_Access := 'TRUE' }
VERSION : 0.1
   VAR 
      ADIN { S7_SetPoint := 'False'} : Array[0.."M_ADIN"] of "AFB_ADIN_v3";
      AIN { S7_SetPoint := 'False'} : Array[0.."M_AIN"] of "AFB_AIN_v3";
      DIFF { S7_SetPoint := 'False'} : Array[0.."M_DIFF"] of "AFB_DIFF_v3";
      DIN { S7_SetPoint := 'False'} : Array[0.."M_DIN"] of "AFB_DIN_v3";
      MTR { S7_SetPoint := 'False'} : Array[0.."M_MTR"] of "AFB_MotorPID_v3";
      MTRLIN { S7_SetPoint := 'False'} : Array[0.."M_MTRLIN"] of "AFB_MotorLinearCtrl_v3";
      MTRDIR { S7_SetPoint := 'False'} : Array[0.."M_MTRDIR"] of "AFB_MotorDirect_v3";
      VLV { S7_SetPoint := 'False'} : Array[0.."M_VLV"] of "AFB_Valve_v3";
      CVLV { S7_SetPoint := 'False'} : Array[0.."M_CVLV"] of "AFB_ControlValve_v3";
   END_VAR

   VAR_TEMP 
      i : Int;
   END_VAR


BEGIN
	FOR #i := 0 TO "M_ADIN" DO
	    
	    "Proc_ADIN"(i := #i,
	                module := #ADIN[#i]);
	    
	END_FOR;
	
	FOR #i := 0 TO "M_AIN" DO
	    
	    "Proc_AIN"(i := #i,
	               module := #AIN[#i]);
	    
	END_FOR;
	
	FOR #i := 0 TO "M_DIFF" DO
	    
	    
	    "Proc_DIFF"(i := #i,
	                module := #DIFF[#i]);
	    
	    
	END_FOR;
	
	FOR #i := 0 TO "M_DIN" DO
	    
	    "Proc_DIN"(i := #i,
	               module := #DIN[#i]);
	    
	END_FOR;
	
	FOR #i := 0 TO "M_MTR" DO
	    
	    
	    "Proc_MTR"(i := #i,
	               module := #MTR[#i]);
	    
	    
	END_FOR;
	
	FOR #i := 0 TO "M_MTRDIR" DO
	    
	    
	    "Proc_MTRDIR"(i := #i,
	                  module := #MTRDIR[#i]);
	    
	    
	END_FOR;
	
	FOR #i := 0 TO "M_MTRLIN" DO
	    
	    "Proc_MTRLIN"(i := #i,
	                  module := #MTRLIN[#i]);
	    
	               END_FOR;
	
	FOR #i := 0 TO "M_VLV" DO
	    
	    "Proc_VLV"(i := #i,
	               module := #VLV[#i]);
	    
	END_FOR;
	
	FOR #i := 0 TO "M_CVLV" DO
	    
	    "Proc_CVLV"(i := #i,
	                module := #CVLV[#i]);
	    
	END_FOR;
END_FUNCTION_BLOCK

FUNCTION "Proc_ADIN" : Void
{ S7_Optimized_Access := 'TRUE' }
VERSION : 0.1
   VAR_INPUT 
      i : Int;
   END_VAR

   VAR_IN_OUT 
      module : "AFB_ADIN_v3";
   END_VAR

   VAR_TEMP 
      indexLEFT : Int;   //  Index for the primary array of module faults
      indexRIGHT : Int;   //  Index for the secondary array of module faults
   END_VAR


BEGIN
	IF "DB_System".modulesGroup.ADIN AND "MODULES_CTRL".ADIN[#i].status THEN
	    
	    // PI: INPUT
	    
	    // IMPLICIT INPUT
	    
	    #module.p1s := "p1s";
	    #module.p100ms := "p100ms";
	    #module.generalackn := "generalAckn";
	    #module.reset := "ResetFaults";
	    #module.mute := "MuteHorn";
	    
	    // EXPLICIT INPUT
	    
	    "explicitInput_ADIN"(i:=#i,
	                         module:=#module);
	    
	    // Run Module
	    
	    #indexLEFT := #i / 8; // decide the type array member
	    
	    IF (#indexLEFT > "MAX_DIN") OR (#indexLEFT < 0) THEN // "IF" has a protective AND NOT corrective role
	         #indexLEFT := "MAX_DIN";
	    END_IF;
	    #indexRIGHT := #i - #indexLEFT * 8; // decide the alarm member inside the previous index
	    
	    IF (#indexRIGHT > 7) THEN // "IF" has a protective and not corrective role
	         #indexRIGHT := 7;
	    END_IF;
	    
	    #module(alarm_adin:="FAULTS".ADIN[#indexLEFT].ctrl[#indexRIGHT],
	            plcackn_adin:="FAULTS".ADIN[#indexLEFT+ 8].ctrl[#indexRIGHT+8],
	            siren_adin:="FAULTS".ADIN[#indexLEFT].status[#indexRIGHT],
	            hmiackn_adin:="FAULTS".ADIN[#indexLEFT +8].status[#indexRIGHT +8]);
	    
	    // EXPLICIT OUTPUT
	    
	    "explicitOutput_ADIN"(i:=#i,
	                          module:=#module);
	    
	ELSE
	    
	    #module.Switch:= FALSE;
	    
	END_IF;
END_FUNCTION

FUNCTION "explicitInput_ADIN" : Void
{ S7_Optimized_Access := 'TRUE' }
VERSION : 0.1
   VAR_INPUT 
      i : Int;
   END_VAR

   VAR_IN_OUT 
      module : "AFB_ADIN_v3";
   END_VAR


BEGIN
	CASE #i OF
	        
	    -1:
	        ;
	        
	    ELSE
	        ;
	END_CASE;
END_FUNCTION

FUNCTION "explicitOutput_ADIN" : Void
{ S7_Optimized_Access := 'TRUE' }
VERSION : 0.1
   VAR_INPUT 
      i : Int;
   END_VAR

   VAR_IN_OUT 
      module : "AFB_ADIN_v3";
   END_VAR


BEGIN
	CASE #i OF
	    -1:
	        ;
	    ELSE
	        ;
	END_CASE;
END_FUNCTION

FUNCTION "Proc_AIN" : Void
{ S7_Optimized_Access := 'TRUE' }
VERSION : 0.1
   VAR_INPUT 
      i : Int;
   END_VAR

   VAR_IN_OUT 
      module : "AFB_AIN_v3";
   END_VAR


BEGIN
	IF "DB_System".modulesGroup.AIN AND "MODULES_CTRL".AIN[#i].status THEN
	    
	    // PI: INPUT
	    
	    // IMPLICIT INPUT
	    
	    #module.reset := "ResetFaults";
	    #module.p1s := "p1s";
	    #module.p100ms := "p100ms";
	    #module.generalackn := "generalAckn";
	    #module.mute := "MuteHorn";
	    #module.t_sys := "DB_System".datetime.current;
	    
	    // EXPLICIT INPUT
	    
	    "explicitInput_AIN"(i:=#i,
	                        module:=#module);
	    
	    // Run Module
	    
	    #module(faults:="FAULTS".AIN[#i],
	            warnings:="WARNINGS".AIN[#i]);
	    
	    // EXPLICIT OUTPUT
	    
	    "explicitOutput_AIN"(i:=#i,
	                         module:=#module);
	    
	ELSE
	    
	    #module.output := 0;
	    
	END_IF;
END_FUNCTION

FUNCTION "explicitInput_AIN" : Void
{ S7_Optimized_Access := 'TRUE' }
VERSION : 0.1
   VAR_INPUT 
      i : Int;
   END_VAR

   VAR_IN_OUT 
      module : "AFB_AIN_v3";
   END_VAR


BEGIN
	CASE #i OF
	        
	    -1:
	        ;
	        
	    ELSE
	        ;
	
	END_CASE;
END_FUNCTION

FUNCTION "explicitOutput_AIN" : Void
{ S7_Optimized_Access := 'TRUE' }
VERSION : 0.1
   VAR_INPUT 
      i : Int;
   END_VAR

   VAR_IN_OUT 
      module : "AFB_AIN_v3";
   END_VAR


BEGIN
	CASE #i OF
	    -1:
	        ;
	    ELSE
	        ;
	END_CASE;
END_FUNCTION

FUNCTION "Proc_DIFF" : Void
{ S7_Optimized_Access := 'TRUE' }
VERSION : 0.1
   VAR_INPUT 
      i : Int;
   END_VAR

   VAR_IN_OUT 
      module : "AFB_DIFF_v3";
   END_VAR


BEGIN
	IF "DB_System".modulesGroup.DIFF AND "MODULES_CTRL".DIFF[#i].status THEN
	    
	    #module.generalackn := "generalAckn";
	    #module.reset := "ResetFaults";
	    #module.mute := "MuteHorn";
	    #module.p1s := "p1s";
	    #module.p100ms := "p100ms";
	    
	    // EXPLICIT INPUT
	    
	    "explicitInput_DIFF"(i:=#i,
	                         module:=#module);
	    
	    // Run Module
	    
	    #module(faults := "FAULTS".AIN[#i],
	            warnings := "WARNINGS".AIN[#i]);
	    
	    // EXPLICIT OUTPUT
	    
	    "explicitOutput_DIFF"(i:=#i,
	                          module:=#module);
	    
	ELSE
	    
	    #module.output := 0;
	    
	END_IF;
END_FUNCTION

FUNCTION "explicitInput_DIFF" : Void
{ S7_Optimized_Access := 'TRUE' }
VERSION : 0.1
   VAR_INPUT 
      i : Int;
   END_VAR

   VAR_IN_OUT 
      module : "AFB_DIFF_v3";
   END_VAR


BEGIN
	CASE #i OF
	    -1:
	        ;
	    ELSE
	        ;
	END_CASE;
END_FUNCTION

FUNCTION "explicitOutput_DIFF" : Void
{ S7_Optimized_Access := 'TRUE' }
VERSION : 0.1
   VAR_INPUT 
      i : Int;
   END_VAR

   VAR_IN_OUT 
      module : "AFB_DIFF_v3";
   END_VAR


BEGIN
	CASE #i OF
	    -1:
	        ;
	    ELSE
	        ;
	END_CASE;
END_FUNCTION

FUNCTION "Proc_DIN" : Void
{ S7_Optimized_Access := 'TRUE' }
VERSION : 0.1
   VAR_INPUT 
      i : Int;
   END_VAR

   VAR_IN_OUT 
      module : "AFB_DIN_v3";
   END_VAR

   VAR_TEMP 
      indexLEFT : Int;   //  Index for the primary array of module faults
      indexRIGHT : Int;   //  Index for the secondary array of module faults
   END_VAR


BEGIN
	IF "DB_System".modulesGroup.DIN AND "MODULES_CTRL".DIN[#i].status THEN
	    
	    // PI: INPUT
	    
	    
	    // IMPLICIT INPUT
	    
	    #module.p1s := "p1s";
	    #module.p100ms := "p100ms";
	    #module.generalackn := "generalAckn";
	    #module.reset := "ResetFaults";
	    #module.mute := "MuteHorn";
	    
	    // EXPLICIT INPUT
	    
	    "explicitInput_DIN"(i:=#i,
	                        module:=#module);
	
	    // Run Module
	    
	    #indexLEFT := #i/8; // decide the type array member
	    
	    IF (#indexLEFT > "MAX_DIN") OR (#indexLEFT < 0) THEN // "IF" has a protective AND NOT corrective role
	         #indexLEFT := "MAX_DIN";
	    END_IF;
	    #indexRIGHT := #i - #indexLEFT * 8; // decide the alarm member inside the previous index
	    
	    IF (#indexRIGHT > 7) THEN // "IF" has a protective and not corrective role
	         #indexRIGHT := 7;
	    END_IF;
	    
	    #module(alarm_din:="FAULTS".DIN[#indexLEFT].ctrl[#indexRIGHT],
	            plcackn_din:="FAULTS".DIN[#indexLEFT+ 8].ctrl[#indexRIGHT+8],
	            siren_din:="FAULTS".DIN[#indexLEFT].status[#indexRIGHT],
	            hmiackn_din:="FAULTS".DIN[#indexLEFT +8].status[#indexRIGHT +8]);
	     
	    // EXPLICIT OUTPUT
	    
	    "explicitOutput_DIN"(i:=#i,
	                         module:=#module);
	    
	ELSE
	    
	    #module.Switch := FALSE;
	    
	END_IF;
END_FUNCTION

FUNCTION "explicitInput_DIN" : Void
{ S7_Optimized_Access := 'TRUE' }
VERSION : 0.1
   VAR_INPUT 
      i : Int;
   END_VAR

   VAR_IN_OUT 
      module : "AFB_DIN_v3";
   END_VAR


BEGIN
	CASE #i OF
	        
	    -1:
	        ;
	        
	    ELSE
	        ;
	END_CASE;
END_FUNCTION

FUNCTION "explicitOutput_DIN" : Void
{ S7_Optimized_Access := 'TRUE' }
VERSION : 0.1
   VAR_INPUT 
      i : Int;
   END_VAR

   VAR_IN_OUT 
      module : "AFB_DIN_v3";
   END_VAR


BEGIN
	CASE #i OF
	    -1:
	        ;
	    ELSE
	        ;
	END_CASE;
END_FUNCTION

FUNCTION "Proc_MTR" : Void
{ S7_Optimized_Access := 'TRUE' }
VERSION : 0.1
   VAR_INPUT 
      i : Int;
   END_VAR

   VAR_IN_OUT 
      module : "AFB_MotorPID_v3";
   END_VAR


BEGIN
	IF "DB_System".modulesGroup.MTR AND "MODULES_CTRL".MTR[#i].status THEN
	    
	    // PI: INPUT
	    
	    
	    // IMPLICIT INPUT
	    
	    #module.generalackn := "generalAckn";
	    #module.reset := "ResetFaults";
	    #module.mute := "MuteHorn";
	    #module.autoset := "AutoSET";
	    #module.manualset := "ManualSET";
	    #module.p1s := "p1s";
	    #module.p100ms := "p100ms";
	    #module.blink := "blink";
	    
	    // EXPLICIT INPUT
	    
	    "explicitInput_MTR"(i:=#i,
	                        module:=#module);
	    
	    // Run Module
	    
	    #module(faults:="FAULTS".MTR[#i]);
	    
	    // PI: OUTPUT
	    
	    
	    // EXPLICIT OUTPUT
	    
	    "explicitOutput_MTR"(i:=#i,
	                         module:=#module);
	    
	ELSE
	    
	    #module.run := FALSE;
	    #module.reference := 0;
	    
	END_IF;
END_FUNCTION

FUNCTION "explicitInput_MTR" : Void
{ S7_Optimized_Access := 'TRUE' }
VERSION : 0.1
   VAR_INPUT 
      i : Int;
   END_VAR

   VAR_IN_OUT 
      module : "AFB_MotorPID_v3";
   END_VAR

   VAR_TEMP 
      reset : Bool;
   END_VAR


BEGIN
	CASE #i OF
	        
	    -1:
	        ;
	        
	    ELSE
	        ;
	END_CASE;
END_FUNCTION

FUNCTION "explicitOutput_MTR" : Void
{ S7_Optimized_Access := 'TRUE' }
VERSION : 0.1
   VAR_INPUT 
      i : Int;
   END_VAR

   VAR_IN_OUT 
      module : "AFB_MotorPID_v3";
   END_VAR


BEGIN
	CASE #i OF
	        
	    -1:
	        ;
	        
	    ELSE
	        ;
	END_CASE;
END_FUNCTION

FUNCTION "Proc_MTRDIR" : Void
{ S7_Optimized_Access := 'TRUE' }
VERSION : 0.1
   VAR_INPUT 
      i : Int;
   END_VAR

   VAR_IN_OUT 
      module : "AFB_MotorDirect_v3";
   END_VAR


BEGIN
	IF "DB_System".modulesGroup.MTRDIR AND "MODULES_CTRL".MTRDIR[#i].status THEN
	    
	    // PI: INPUT
	   
	    
	    // IMPLICIT INPUT
	    
	    #module.generalackn := "generalAckn";
	    #module."reset" := "ResetFaults";
	    #module.mute := "MuteHorn";
	    #module."autoset" := "AutoSET";
	    #module."manualset" := "ManualSET";
	    #module.p1s := "p1s";
	    #module.p100ms := "p100ms";
	    #module.blink := "blink";
	    
	    //#module.block := "EMERGENCY";
	    
	    // EXPLICIT INPUT
	    
	    "explicitInput_MTRDIR"(i:=#i,
	                           module:=#module);
	    
	    // Run Module
	    
	    #module(faults := "FAULTS".MTRDIR[#i]);
	    
	    // PI: OUTPUT
	    
	    
	    // EXPLICIT OUTPUT
	    
	    "explicitOutput_MTRDIR"(i:=#i,
	                            module:=#module);
	    
	ELSE
	    
	    #module.run := FALSE;
	    
	
	    
	END_IF;
END_FUNCTION

FUNCTION "explicitInput_MTRDIR" : Void
{ S7_Optimized_Access := 'TRUE' }
VERSION : 0.1
   VAR_INPUT 
      i : Int;
   END_VAR

   VAR_IN_OUT 
      module : "AFB_MotorDirect_v3";
   END_VAR


BEGIN
	CASE #i OF
	        
	    -1:
	        ;
	        
	    ELSE
	        ;
	END_CASE;
END_FUNCTION

FUNCTION "explicitOutput_MTRDIR" : Void
{ S7_Optimized_Access := 'TRUE' }
VERSION : 0.1
   VAR_INPUT 
      i : Int;
   END_VAR

   VAR_IN_OUT 
      module : "AFB_MotorDirect_v3";
   END_VAR


BEGIN
	CASE #i OF
	        
	    -1:
	        ;
	        
	    ELSE
	        ;
	END_CASE;
END_FUNCTION

FUNCTION "Proc_MTRLIN" : Void
{ S7_Optimized_Access := 'TRUE' }
VERSION : 0.1
   VAR_INPUT 
      i : Int;
   END_VAR

   VAR_IN_OUT 
      module : "AFB_MotorLinearCtrl_v3";
   END_VAR


BEGIN
	IF "DB_System".modulesGroup.MTRLIN AND "MODULES_CTRL".MTRLIN[#i].status THEN
	    
	    // PI: INPUT
	    
	    
	    // IMPLICIT INPUT
	    
	    #module."reset" := "ResetFaults";
	    #module."autoset" := "AutoSET";
	    #module."manualset" := "ManualSET";
	    #module.p1s := "p1s";
	    #module.p100ms := "p100ms";
	    #module.generalackn := "generalAckn";
	    #module.mute := "MuteHorn";
	    #module.blink := "blink";
	    
	    //#module.block := "EMERGENCY";
	    
	    // EXPLICIT INPUT
	    
	    "explicitInput_MTRLIN"(i:=#i,
	                           module:=#module);
	    
	    
	    // Run Module
	    
	    #module(faults := "FAULTS".MTRLIN[#i]);
	    
	    // PI: OUTPUT
	    
	    
	    // EXPLICIT OUTPUT
	    
	    "explicitOutput_MTRLIN"(i:=#i,
	                            module:=#module);
	    
	ELSE
	    
	    #module.run:= FALSE;
	    #module.reference := 0;
	    
	    
	END_IF;
END_FUNCTION

FUNCTION "explicitInput_MTRLIN" : Void
{ S7_Optimized_Access := 'TRUE' }
VERSION : 0.1
   VAR_INPUT 
      i : Int;
   END_VAR

   VAR_IN_OUT 
      module : "AFB_MotorLinearCtrl_v3";
   END_VAR


BEGIN
	CASE #i OF
	        
	    -1:
	        ;
	        
	    ELSE
	        ;
	END_CASE;
END_FUNCTION

FUNCTION "explicitOutput_MTRLIN" : Void
{ S7_Optimized_Access := 'TRUE' }
VERSION : 0.1
   VAR_INPUT 
      i : Int;
   END_VAR

   VAR_IN_OUT 
      module : "AFB_MotorLinearCtrl_v3";
   END_VAR


BEGIN
	CASE #i OF
	    -1:
	        ;
	    ELSE
	        ;
	END_CASE;
END_FUNCTION

FUNCTION "Proc_VLV" : Void
{ S7_Optimized_Access := 'TRUE' }
VERSION : 0.1
   VAR_INPUT 
      i : Int;
   END_VAR

   VAR_IN_OUT 
      module : "AFB_Valve_v3";
   END_VAR


BEGIN
	IF "DB_System".modulesGroup.VLV AND "MODULES_CTRL".VLV[#i].status THEN
	    
	    // PI: INPUT
	    
	    
	    // IMPLICIT INPUT
	
	    #module.generalackn := "generalAckn";
	    #module."reset" := "ResetFaults";
	    #module.mute := "MuteHorn";
	    #module."autoset" := "AutoSET";
	    #module."manualset" := "ManualSET";
	    #module.p1s := "p1s";
	    #module.p100ms := "p100ms";
	    #module.blink := "blink";
	    
	    // EXPLICIT INPUT
	    
	    "explicitInput_VLV"(i:=#i,
	                        module:=#module);
	    
	    
	    // Run Module
	    
	    #module(faults:="FAULTS".VLV[#i]);
	    
	    // PI: OUTPUT
	    
	    
	    // EXPLICIT OUTPUT
	    
	    "explicitOutput_VLV"(i:=#i,
	                         module:=#module);
	    
	ELSE
	    
	    #module.main:=FALSE;
	    #module.upper := FALSE;
	    #module.lower := FALSE;
	    
	    
	END_IF;
END_FUNCTION

FUNCTION "explicitInput_VLV" : Void
{ S7_Optimized_Access := 'TRUE' }
VERSION : 0.1
   VAR_INPUT 
      i : Int;
   END_VAR

   VAR_IN_OUT 
      module : "AFB_Valve_v3";
   END_VAR


BEGIN
	CASE #i OF
	        
	    -1:
	        ;
	        
	    ELSE
	        ;
	END_CASE;
END_FUNCTION

FUNCTION "explicitOutput_VLV" : Void
{ S7_Optimized_Access := 'TRUE' }
VERSION : 0.1
   VAR_INPUT 
      i : Int;
   END_VAR

   VAR_IN_OUT 
      module : "AFB_Valve_v3";
   END_VAR


BEGIN
	CASE #i OF
	        
	    -1:
	        ;
	        
	    ELSE
	        ;
	END_CASE;
END_FUNCTION

FUNCTION "Proc_CVLV" : Void
{ S7_Optimized_Access := 'TRUE' }
VERSION : 0.1
   VAR_INPUT 
      i : Int;
   END_VAR

   VAR_IN_OUT 
      module : "AFB_ControlValve_v3";
   END_VAR


BEGIN
	IF "DB_System".modulesGroup.CVLV AND "MODULES_CTRL".CVLV[#i].status THEN
	    
	    // IMPLICIT INPUT
	    
	    #module.p1s := "p1s";
	    #module.p100ms := "p100ms";
	    #module.blink := "blink";
	    
	    // EXPLICIT INPUT
	    
	    "explicitInput_CVLV"(i:=#i,
	                         module:=#module);
	    
	    // Run Module
	    
	    #module();
	    
	    // PI: OUTPUT
	    
	    
	    // EXPLICIT OUTPUT
	    
	    "explicitOutput_CVLV"(i:=#i,
	                          module:=#module);
	    
	ELSE
	    
	    #module.reference := 0;
	    
	    
	END_IF;
END_FUNCTION

FUNCTION "explicitInput_CVLV" : Void
{ S7_Optimized_Access := 'TRUE' }
VERSION : 0.1
   VAR_INPUT 
      i : Int;
   END_VAR

   VAR_IN_OUT 
      module : "AFB_ControlValve_v3";
   END_VAR


BEGIN
	CASE #i OF
	    -1:
	        ;
	        
	    ELSE
	        ;
	END_CASE;
END_FUNCTION

FUNCTION "explicitOutput_CVLV" : Void
{ S7_Optimized_Access := 'TRUE' }
VERSION : 0.1
   VAR_INPUT 
      i : Int;
   END_VAR

   VAR_IN_OUT 
      module : "AFB_ControlValve_v3";
   END_VAR


BEGIN
	CASE #i OF
	    -1:
	        ;
	    ELSE
	        ;
	END_CASE;
END_FUNCTION

FUNCTION_BLOCK "AFB_ResetModules"
{ S7_Optimized_Access := 'TRUE' }
VERSION : 0.1
   VAR 
      c_vlv : "C_VLV";
      c_cvlv : "C_CVLV";
      c_mtr : "C_MTR";
      c_mtrdir : "C_MTRDIR";
      c_mtrlin : "C_MTRLIN";
   END_VAR

   VAR_TEMP 
      i : Int;
   END_VAR


BEGIN
	FOR #i := 0 TO "M_CVLV" DO
	    
	    #c_cvlv(enable := TRUE,
	           index := #i,
	           cmd := FALSE,
	           fup:=FALSE);
	    
	END_FOR;
	
	FOR #i := 0 TO "M_VLV" DO
	    
	    #c_vlv(enable := TRUE,
	           index := #i,
	           cmd := FALSE,
	           upper:=FALSE,
	           lower:=FALSE);
	    
	END_FOR;
	
	FOR #i := 0 TO "M_MTR" DO
	    
	    #c_mtr(enable := TRUE,
	           index := #i,
	           cmd := FALSE,
	           followUp:=FALSE);
	    
	END_FOR;
	
	FOR #i := 0 TO "M_MTRDIR" DO
	    
	    #c_mtrdir(enable := TRUE,
	           index := #i,
	           cmd := FALSE);
	    
	END_FOR;
	
	FOR #i := 0 TO "M_MTRLIN" DO
	     
	     #c_mtrlin(enable := TRUE,
	               index := #i,
	               cmd := FALSE,
	               fup:=FALSE);
	     
	END_FOR;
END_FUNCTION_BLOCK

FUNCTION_BLOCK "C_VLV"
{ S7_Optimized_Access := 'TRUE' }
VERSION : 0.1
   VAR_INPUT 
      enable { ExternalAccessible := 'False'; ExternalVisible := 'False'; ExternalWritable := 'False'} : Bool;   //  TRUE: Enable module
      index : Int;   //  INDEX
      cmd : Bool;   //  TRUE: Activate main
      upper : Bool;   //  TRUE: Activate upper
      lower : Bool;   //  TRUE: Activate lower
      blockMain : Bool;   //  TRUE: Block main activation
      blockUpper : Bool;   //  TRUE: Block upper activation
      blockLower : Bool;   //  TRUE: Block lower activation
   END_VAR

   VAR_OUTPUT 
      vfbMain { ExternalAccessible := 'False'; ExternalVisible := 'False'; ExternalWritable := 'False'} : Bool;
      hasJustAct { ExternalAccessible := 'False'; ExternalVisible := 'False'; ExternalWritable := 'False'} : Bool;
      vfbDeact { ExternalAccessible := 'False'; ExternalVisible := 'False'; ExternalWritable := 'False'} : Bool;
      hasjustDeact { ExternalAccessible := 'False'; ExternalVisible := 'False'; ExternalWritable := 'False'} : Bool;
      fault { ExternalAccessible := 'False'; ExternalVisible := 'False'; ExternalWritable := 'False'} : Bool;
      justHadFault { ExternalAccessible := 'False'; ExternalVisible := 'False'; ExternalWritable := 'False'} : Bool;
      justLostFault { ExternalAccessible := 'False'; ExternalVisible := 'False'; ExternalWritable := 'False'} : Bool;
      enabled { ExternalAccessible := 'False'; ExternalVisible := 'False'; ExternalWritable := 'False'} : Bool;
      auto { ExternalAccessible := 'False'; ExternalVisible := 'False'; ExternalWritable := 'False'} : Bool;
   END_VAR

   VAR 
      status { ExternalAccessible := 'False'; ExternalVisible := 'False'; ExternalWritable := 'False'; S7_SetPoint := 'False'} : "UDT_STATUS_VLV";
   END_VAR

   VAR_TEMP 
      module : "UDT_VALVE";
      resetStatus : "UDT_STATUS_VLV";
   END_VAR


BEGIN
	
	
	IF #enable THEN
	     
	     #status.enabled := TRUE;
	     
	     #module := "MOD".VLV[#index].i;
	     
	     REGION STATUS
	          
	          #status.isAct := #module.status.vfbmain;
	          #status.inFault := #module.status.fault;
	          
	          #status.hasJustAct := "detectPE"(newValue := #status.isAct, oldValue := #status.old.position);
	          #status.hasjustDeact := "detectNE"(newValue := #status.isAct, oldValue := #status.old.position);
	          #status.justHadFault := "detectPE"(newValue := #status.inFault, oldValue := #status.old.fault);
	          #status.justLostFault := "detectNE"(newValue := #status.inFault, oldValue := #status.old.fault);
	          
	          #status.auto := #module.ind.auto;
	          
	          #status.old.position := #status.isAct;
	          #status.old.fault := #status.inFault;
	          
	     END_REGION
	     
	     REGION COMMAND
	          
	          "MOD".VLV[#index].actmain := #cmd;
	          "MOD".VLV[#index].actupper := #upper;
	          "MOD".VLV[#index].actlower := #lower;
	          "MOD".VLV[#index].blockmain := #blockMain;
	          "MOD".VLV[#index].blockupper := #blockUpper;
	          "MOD".VLV[#index].blocklower := #blockLower;
	          
	          
	     END_REGION
	     
	     REGION SIM
	          
	          // "MOD".VLV[#index].i.sim.main := "MODULES_CTRL".VLV[#index].sim.simMain AND NOT "MODULES_CTRL".VLV[#index].sim.simDeact;
	          // "MOD".VLV[#index].i.sim.upper := "MODULES_CTRL".VLV[#index].sim.simLower;
	          // "MOD".VLV[#index].i.sim.lower := "MODULES_CTRL".VLV[#index].sim.simUpper;
	          // "MOD".VLV[#index].i.sim.deact := "MODULES_CTRL".VLV[#index].sim.simDeact;
	          
	     END_REGION
	     
	ELSE
	    ;
	     // #status := #resetStatus;
	     
	     // "MOD".VLV[#index].actmain := FALSE;
	     // "MOD".VLV[#index].actupper := FALSE;
	     // "MOD".VLV[#index].actlower := FALSE;
	     // "MOD".VLV[#index].blockmain := FALSE;
	     // "MOD".VLV[#index].blockupper := FALSE;
	     // "MOD".VLV[#index].blocklower := FALSE;
	     
	END_IF;
	
	REGION Output
	     
	     #vfbMain := #status.isAct;
	     #hasJustAct := #status.hasJustAct;
	     #vfbDeact := #status.isDeact;
	     #hasjustDeact := #status.hasjustDeact;
	     #fault := #status.inFault;
	     #justHadFault := #status.justHadFault;
	     #justLostFault := #status.justLostFault;
	     #enabled := #status.enabled;
	     #auto := #status.auto;
	     
	END_REGION Output
END_FUNCTION_BLOCK

FUNCTION "detectPE" : Bool
{ S7_Optimized_Access := 'TRUE' }
VERSION : 0.1
   VAR_INPUT 
      newValue : Bool;
      oldValue : Bool;
   END_VAR


BEGIN
	#detectPE := #newValue AND NOT #oldValue;
END_FUNCTION

FUNCTION "detectNE" : Bool
{ S7_Optimized_Access := 'TRUE' }
VERSION : 0.1
   VAR_INPUT 
      newValue : Bool;
      oldValue : Bool;
   END_VAR


BEGIN
	#detectNE := NOT #newValue AND #oldValue;
END_FUNCTION

FUNCTION_BLOCK "C_CVLV"
{ S7_Optimized_Access := 'TRUE' }
VERSION : 0.1
   VAR_INPUT 
      enable { ExternalAccessible := 'False'; ExternalVisible := 'False'; ExternalWritable := 'False'} : Bool;
      index : Int;
      cmd : Bool;
      fup : Bool;
   END_VAR

   VAR 
      status { ExternalAccessible := 'False'; ExternalVisible := 'False'; ExternalWritable := 'False'; S7_SetPoint := 'False'} : "UDT_STATUS_CVLV";
   END_VAR

   VAR_TEMP 
      module : "UDT_CONTROLVALVE";
      resetStatus : "UDT_STATUS_CVLV";
   END_VAR


BEGIN
	IF #enable THEN
	    
	    #status.enabled := TRUE;
	    
	    #module := "MOD".CVLV[#index].i;
	    
	    REGION STATUS
	        
	         #status.running := #module.out.vfbact;
	        
	        #status.reference := #module.out."ref";
	        
	        #status.justStarted := "detectPE"(newValue := #status.running, oldValue := #status.old.running);
	        #status.justStopped := "detectNE"(newValue := #status.running, oldValue := #status.old.running);
	        
	        #status.old.running := #status.running;
	        
	    END_REGION
	    
	    REGION COMMAND
	        
	         "MOD".CVLV[#index].control := #cmd;
	         "MOD".CVLV[#index].followup := #fup;
	         
	        
	    END_REGION
	    
	ELSE
	    
	    #status := #resetStatus;
	    
	    "MOD".CVLV[#index].control := #cmd;
	    "MOD".CVLV[#index].followup := #fup;
	    
	END_IF;
END_FUNCTION_BLOCK

FUNCTION_BLOCK "C_MTR"
{ S7_Optimized_Access := 'TRUE' }
VERSION : 0.1
   VAR_INPUT 
      enable { ExternalAccessible := 'False'; ExternalVisible := 'False'; ExternalWritable := 'False'} : Bool;   //  TRUE: Enable module
      index : Int;   //  INDEX
      cmd : Bool;   //  TRUE: Activate main
      block : Bool;   //  TRUE: Block activation
      followUp : Bool;   //  TRUE: Follow-up
      spSource : Bool;   //  TRUE: External setpoint
      FUP : Real;   //  Follow up speed
      SP : Real;   //  SP for PID control
      PV : Real;   //  PV for PID control
      PVunit : WString;   //  Unit of PID PV
   END_VAR

   VAR_OUTPUT 
      vfb : Bool;
      fault : Bool;
      justStarted : Bool;
      justStopped : Bool;
      justHadFault : Bool;
      justLostFault : Bool;
      enabled : Bool;
      auto : Bool;
   END_VAR

   VAR 
      status { ExternalAccessible := 'False'; ExternalVisible := 'False'; ExternalWritable := 'False'; S7_SetPoint := 'False'} : "UDT_STATUS_MTR";
   END_VAR

   VAR_TEMP 
      module : "UDT_MOTOR";
      resetStatus : "UDT_STATUS_MTR";
   END_VAR


BEGIN
	IF #enable THEN
	    
	    #status.enabled := TRUE;
	    
	    #module := "MOD".MTR[#index].i;
	    
	    REGION STATUS
	        
	        #status.running := #module.status.vfb;
	        #status.inFault := #module.status.fault;
	        #status.auto := #module.ind.auto;
	        
	        #status.justStarted := "detectPE"(newValue := #status.running, oldValue := #status.old.running);
	        #status.justStopped := "detectNE"(newValue := #status.running, oldValue := #status.old.running);
	        #status.justHadFault := "detectPE"(newValue := #status.inFault, oldValue := #status.old.fault);
	        #status.justLostFault := "detectNE"(newValue := #status.inFault, oldValue := #status.old.fault);
	        
	        #status.old.running := #status.running;
	        #status.old.fault := #status.inFault;
	        
	
	        
	    END_REGION
	    
	    REGION COMMAND
	        
	        "MOD".MTR[#index].start := #cmd;
	         "MOD".MTR[#index].block := #"block";
	         "MOD".MTR[#index].followup := #"followUp";
	         "MOD".MTR[#index].spsource := #spSource;
	         
	         "MOD".MTR[#index].FUP := #FUP;
	         "MOD".MTR[#index].EXT_SP := #SP;
	         "MOD".MTR[#index].PV := #PV;
	         "MOD".MTR[#index].PV_unit := #PVunit;
	         
	         
	    END_REGION
	    
	    REGION SIM
	        
	        "MOD".MTR[#index].i.sim.fb := "MODULES_CTRL".MTR[#index].sim.simFb;
	        "MOD".MTR[#index].i.sim.ctrl := "MODULES_CTRL".MTR[#index].sim.simCtrl;
	        
	    END_REGION
	    
	ELSE
	    
	    #status := #resetStatus;
	    
	    "MOD".MTR[#index].start := FALSE;
	    "MOD".MTR[#index].block := FALSE;
	    "MOD".MTR[#index].followup := FALSE;
	    "MOD".MTR[#index].spsource := FALSE;
	    
	END_IF;
	
	REGION Output
	    
	    #vfb:= #status.running;
	    #justStarted := #status.justStarted;
	    #justStopped := #status.justStopped;
	    #fault := #status.inFault;
	    #justHadFault := #status.justHadFault;
	    #justLostFault := #status.justLostFault;
	    #enabled := #status.enabled;
	    #auto := #status.auto;
	    
	END_REGION Output
END_FUNCTION_BLOCK

FUNCTION_BLOCK "C_MTRDIR"
{ S7_Optimized_Access := 'TRUE' }
VERSION : 0.1
   VAR_INPUT 
      enable { ExternalAccessible := 'False'; ExternalVisible := 'False'; ExternalWritable := 'False'} : Bool;
      index : Int;
      cmd : Bool;
   END_VAR

   VAR 
      status { ExternalAccessible := 'False'; ExternalVisible := 'False'; ExternalWritable := 'False'; S7_SetPoint := 'False'} : "UDT_STATUS_MTRDIR";
   END_VAR

   VAR_TEMP 
      module : "UDT_MOTORDIRECT";
      resetStatus : "UDT_STATUS_MTRDIR";
   END_VAR


BEGIN
	IF #enable THEN
	    
	    #status.enabled := TRUE;
	    
	    #module := "MOD".MTRDIR[#index].i;
	    
	    REGION STATUS
	        
	        #status.running := #module.status.vfb;
	        
	        #status.justStarted := "detectPE"(newValue := #status.running, oldValue := #status.old.running);
	        #status.justStopped := "detectNE"(newValue := #status.running, oldValue := #status.old.running);
	        #status.justHadFault := "detectPE"(newValue := #status.inFault, oldValue := #status.old.fault);
	        #status.justLostFault := "detectNE"(newValue := #status.inFault, oldValue := #status.old.fault);
	        
	        #status.old.running := #status.running;
	        #status.old.fault := #status.inFault;
	        
	    END_REGION
	    
	    REGION COMMAND
	        
	        "MOD".MTRDIR[#index].start := #cmd;
	        
	    END_REGION
	    
	    REGION SIM
	        
	        "MOD".MTRDIR[#index].i.sim.fb := "MODULES_CTRL".MTRDIR[#index].sim.simFb;
	        "MOD".MTRDIR[#index].i.sim.ctrl := "MODULES_CTRL".MTRDIR[#index].sim.simCtrl;
	        
	    END_REGION
	    
	ELSE
	    
	    #status := #resetStatus;
	    
	    "MOD".MTRDIR[#index].start := FALSE;
	    
	END_IF;
END_FUNCTION_BLOCK

FUNCTION_BLOCK "C_MTRLIN"
{ S7_Optimized_Access := 'TRUE' }
VERSION : 0.1
   VAR_INPUT 
      enable { ExternalAccessible := 'False'; ExternalVisible := 'False'; ExternalWritable := 'False'} : Bool;
      index : Int;
      cmd : Bool;
      fup : Bool;
   END_VAR

   VAR 
      status { ExternalAccessible := 'False'; ExternalVisible := 'False'; ExternalWritable := 'False'; S7_SetPoint := 'False'} : "UDT_STATUS_MTRLIN";
   END_VAR

   VAR_TEMP 
      module : "UDT_MOTORLINEAR";
      resetStatus : "UDT_STATUS_MTRLIN";
   END_VAR


BEGIN
	IF #enable THEN
	    
	    #status.enabled := TRUE;
	    
	    #module := "MOD".MTRLIN[#index].i;
	    
	    REGION STATUS
	        
	        #status.running := #module.status.vfb;
	        #status.inFault := #module.status.fault;
	        
	        #status.reference := #module.out."ref";
	        
	        #status.justStarted := "detectPE"(newValue := #status.running, oldValue := #status.old.running);
	        #status.justStopped := "detectNE"(newValue := #status.running, oldValue := #status.old.running);
	        #status.justHadFault := "detectPE"(newValue := #status.inFault, oldValue := #status.old.fault);
	        #status.justLostFault := "detectNE"(newValue := #status.inFault, oldValue := #status.old.fault);
	        
	        #status.old.running := #status.running;
	        #status.old.fault := #status.inFault;
	        
	    END_REGION
	    
	    REGION COMMAND
	        
	         "MOD".MTRLIN[#index].start := #cmd;
	        "MOD".MTRLIN[#index].followup := #fup;
	        
	    END_REGION
	    
	    REGION SIM
	        
	        "MOD".MTRLIN[#index].i.sim.fb := "MODULES_CTRL".MTRLIN[#index].sim.simFb;
	        "MOD".MTRLIN[#index].i.sim.ctrl := "MODULES_CTRL".MTRLIN[#index].sim.simCtrl;
	        
	    END_REGION
	    
	ELSE
	    
	    #status := #resetStatus;
	    
	    "MOD".MTRLIN[#index].start := #cmd;
	    "MOD".MTRLIN[#index].followup := #fup;
	    
	END_IF;
END_FUNCTION_BLOCK

FUNCTION_BLOCK "C_ADIN"
{ S7_Optimized_Access := 'TRUE' }
VERSION : 0.1
   VAR_INPUT 
      enable { ExternalAccessible := 'False'; ExternalVisible := 'False'; ExternalWritable := 'False'} : Bool;
      index : Int;
   END_VAR

   VAR 
      status { ExternalAccessible := 'False'; ExternalVisible := 'False'; ExternalWritable := 'False'; S7_SetPoint := 'False'} : "UDT_STATUS_DIN";
   END_VAR

   VAR_TEMP 
      module : "UDT_ADIN";
      resetStatus : "UDT_STATUS_AIN";
   END_VAR


BEGIN
	IF #enable THEN
	    
	    #status.enabled := TRUE;
	    
	    #module := "MOD".ADIN[#index].i;
	    
	    REGION STATUS
	        
	        #status.switch := #module.status.switch_active;
	        #status.fault := #module.status.fault;
	        
	        #status.justActivated := "detectPE"(newValue := #status.switch, oldValue := #status.old.switch);
	        #status.justDectivated := "detectNE"(newValue := #status.switch, oldValue := #status.old.switch);
	        #status.justHadFault := "detectPE"(newValue := #status.fault, oldValue := #status.old.fault);
	        #status.justLostFault := "detectNE"(newValue := #status.fault, oldValue := #status.old.fault);
	        
	        #status.old.switch := #status.switch;
	        #status.old.fault := #status.fault;
	        
	    END_REGION
	    
	    REGION SIM
	        
	        "MOD".ADIN[#index].i.sim.simulated := "MODULES_CTRL".ADIN[#index].sim."en";
	        "MOD".ADIN[#index].i.sim.forced := "MODULES_CTRL".ADIN[#index].sim.value;
	        
	    END_REGION
	    
	ELSE
	    
	    #status.enabled := FALSE;
	    
	END_IF;
END_FUNCTION_BLOCK

FUNCTION_BLOCK "C_AIN"
{ S7_Optimized_Access := 'TRUE' }
VERSION : 0.1
   VAR_INPUT 
      enable { ExternalAccessible := 'False'; ExternalVisible := 'False'; ExternalWritable := 'False'} : Bool;
      index : Int;
   END_VAR

   VAR_OUTPUT 
      fault : Bool;
      warning : Bool;
      justHadFault : Bool;
      justLostFault : Bool;
      justHadWarning : Bool;
      justLostWarning : Bool;
      enabled : Bool;
      output : Real;
      unit : WString;
   END_VAR

   VAR 
      status { ExternalAccessible := 'False'; ExternalVisible := 'False'; ExternalWritable := 'False'; S7_SetPoint := 'False'} : "UDT_STATUS_AIN";
   END_VAR

   VAR_TEMP 
      module : "UDT_AIN";
      resetStatus : "UDT_STATUS_AIN";
   END_VAR


BEGIN
	IF #enable THEN
	    
	    #status.enabled := TRUE;
	    #module := "MOD".AIN[#index].i;
	    
	    REGION STATUS
	        
	        #status.warning := #module.faults.l.status.alarm;
	        #status.fault := #module.faults.ll.status.alarm;
	        #status.value := #module.output;
	        #status.unit := #module.unit;
	        
	        #status.justHadWarning := "detectPE"(newValue := #status.warning, oldValue := NOT #status.old.warning);
	        #status.justLostWarning := "detectNE"(newValue := #status.warning, oldValue := NOT #status.old.warning);
	        #status.justHadFault := "detectPE"(newValue := #status.fault, oldValue := NOT #status.old.fault);
	        #status.justLostFault := "detectNE"(newValue := #status.fault, oldValue := NOT #status.old.fault);
	        
	        #status.old.fault := #status.fault;
	        #status.old.warning := #status.warning;
	        
	    END_REGION
	    
	    REGION SIM
	        
	        "MOD".AIN[#index].i.sim."en" := "MODULES_CTRL".AIN[#index].sim."en";
	        "MOD".AIN[#index].i.sim.value := "MODULES_CTRL".AIN[#index].sim.value;
	        
	    END_REGION
	    
	ELSE
	    
	    #status := #resetStatus;
	    
	END_IF;
	
	REGION Output
	    
	    #fault := #status.fault;
	    #warning := #status.warning;
	    #justHadFault := #status.justHadFault;
	    #justLostFault := #status.justLostFault;
	    #justHadWarning := #status.justHadWarning;
	    #justLostWarning := #status.justLostWarning;
	    #enabled := #status.enabled;
	    #output := #status.value;
	    #unit := #status.unit;
	    
	END_REGION Output
END_FUNCTION_BLOCK

FUNCTION_BLOCK "C_DIN"
{ S7_Optimized_Access := 'TRUE' }
VERSION : 0.1
   VAR_INPUT 
      enable { ExternalAccessible := 'False'; ExternalVisible := 'False'; ExternalWritable := 'False'} : Bool;
      index : Int;
   END_VAR

   VAR 
      status { ExternalAccessible := 'False'; ExternalVisible := 'False'; ExternalWritable := 'False'; S7_SetPoint := 'False'} : "UDT_STATUS_DIN";
   END_VAR

   VAR_TEMP 
      module : "UDT_DIN";
      resetStatus : "UDT_STATUS_DIN";
   END_VAR


BEGIN
	IF #enable THEN
	    
	    #status.enabled := TRUE;
	    
	    #module := "MOD".DIN[#index].i;
	    
	    REGION STATUS
	        
	        #status.switch := #module.status.switch_active;
	        #status.fault := #module.status.fault;
	        
	        #status.justActivated := "detectPE"(newValue := #status.switch, oldValue := #status.old.switch);
	        #status.justDectivated := "detectNE"(newValue := #status.switch, oldValue := #status.old.switch);
	        #status.justHadFault := "detectPE"(newValue := #status.fault, oldValue := #status.old.fault);
	        #status.justLostFault := "detectNE"(newValue := #status.fault, oldValue := #status.old.fault);
	        
	        #status.old.switch := #status.switch;
	        #status.old.fault := #status.fault;
	        
	    END_REGION
	    
	    REGION SIM
	        
	        "MOD".DIN[#index].i.sim.simulated := "MODULES_CTRL".DIN[#index].sim."en";
	        "MOD".DIN[#index].i.sim.cmdforce := "MODULES_CTRL".DIN[#index].sim.value;
	        
	    END_REGION
	    
	ELSE
	    
	    #status := #resetStatus;
	    
	END_IF;
END_FUNCTION_BLOCK

FUNCTION_BLOCK "pALARMS"
{ S7_Optimized_Access := 'TRUE' }
AUTHOR : CH
FAMILY : Aktina
NAME : Faults
VERSION : 0.1
   VAR 
      "75sf1" { S7_SetPoint := 'False'} : "AFB_AlarmAckn";
   END_VAR


BEGIN
	REGION FAULT
	    
	    //Safety fault: Emergency button 75SF1
	    // #"75sf1"(trigger := NOT "di_Emergency_btn",
	    //          release := TRUE,
	    //          ctrlpoint := TRUE,
	    //          enackn := TRUE,
	    //          ensiren := TRUE,
	    //          p100ms := "p100ms",
	    //          generalackn := "ResetFaults",
	    //          reset := "ResetFaults",
	    //          mute :="MuteHorn",
	    //          delay := 0.5,
	    //          plcackn => "FAULTS".Plant[0].ctrl[8],
	    //          alarm => "FAULTS".Plant[0].ctrl[0],
	    //          siren => "FAULTS".Plant[0].status[0],
	    //          hmiackn := "FAULTS".Plant[0].status[8]);
	    
	
	   
	
	
	END_REGION
	
	REGION WARNING
	    
	     
	END_REGION
END_FUNCTION_BLOCK

DATA_BLOCK "dbSysInfo"   // DB2
AUTHOR : CH
FAMILY : Aktina
NAME : Lib_System
// stored: AutoNumber false, InstanceOfName libCpu_SystemInfo, InstanceOfType FB
"libCpu_SystemInfo"
BEGIN
END_DATA_BLOCK

DATA_BLOCK "ResetModules"   // DB4
// stored: InstanceOfName AFB_ResetModules, InstanceOfType FB
"AFB_ResetModules"
BEGIN
   c_vlv.enable := FALSE;
   c_vlv.index := 0;
   c_vlv.cmd := FALSE;
   c_vlv.upper := FALSE;
   c_vlv.lower := FALSE;
   c_vlv.blockMain := FALSE;
   c_vlv.blockUpper := FALSE;
   c_vlv.blockLower := FALSE;
   c_vlv.vfbMain := FALSE;
   c_vlv.hasJustAct := FALSE;
   c_vlv.vfbDeact := FALSE;
   c_vlv.hasjustDeact := FALSE;
   c_vlv.fault := FALSE;
   c_vlv.justHadFault := FALSE;
   c_vlv.justLostFault := FALSE;
   c_vlv.enabled := FALSE;
   c_vlv.auto := FALSE;
   c_vlv.status.isAct := FALSE;
   c_vlv.status.hasJustAct := FALSE;
   c_vlv.status.isDeact := FALSE;
   c_vlv.status.hasjustDeact := FALSE;
   c_vlv.status.inFault := FALSE;
   c_vlv.status.justHadFault := FALSE;
   c_vlv.status.justLostFault := FALSE;
   c_vlv.status.enabled := FALSE;
   c_vlv.status.auto := FALSE;
   c_vlv.status.old.position := FALSE;
   c_vlv.status.old.fault := FALSE;
   c_cvlv.enable := FALSE;
   c_cvlv.index := 0;
   c_cvlv.cmd := FALSE;
   c_cvlv.fup := FALSE;
   c_cvlv.status.running := FALSE;
   c_cvlv.status.justStarted := FALSE;
   c_cvlv.status.justStopped := FALSE;
   c_cvlv.status.reference := 0.0;
   c_cvlv.status.enabled := FALSE;
   c_cvlv.status.old.running := FALSE;
   c_mtr.enable := FALSE;
   c_mtr.index := 0;
   c_mtr.cmd := FALSE;
   c_mtr.block := FALSE;
   c_mtr.followUp := FALSE;
   c_mtr.spSource := FALSE;
   c_mtr.FUP := 0.0;
   c_mtr.SP := 0.0;
   c_mtr.PV := 0.0;
   c_mtr.PVunit := WSTRING#'';
   c_mtr.vfb := FALSE;
   c_mtr.fault := FALSE;
   c_mtr.justStarted := FALSE;
   c_mtr.justStopped := FALSE;
   c_mtr.justHadFault := FALSE;
   c_mtr.justLostFault := FALSE;
   c_mtr.enabled := FALSE;
   c_mtr.auto := FALSE;
   c_mtr.status.running := FALSE;
   c_mtr.status.inFault := FALSE;
   c_mtr.status.justStarted := FALSE;
   c_mtr.status.justStopped := FALSE;
   c_mtr.status.justHadFault := FALSE;
   c_mtr.status.justLostFault := FALSE;
   c_mtr.status.reference := 0.0;
   c_mtr.status.enabled := FALSE;
   c_mtr.status.auto := FALSE;
   c_mtr.status.old.running := FALSE;
   c_mtr.status.old.fault := FALSE;
   c_mtrdir.enable := FALSE;
   c_mtrdir.index := 0;
   c_mtrdir.cmd := FALSE;
   c_mtrdir.status.running := FALSE;
   c_mtrdir.status.inFault := FALSE;
   c_mtrdir.status.justStarted := FALSE;
   c_mtrdir.status.justStopped := FALSE;
   c_mtrdir.status.justHadFault := FALSE;
   c_mtrdir.status.justLostFault := FALSE;
   c_mtrdir.status.enabled := FALSE;
   c_mtrdir.status.old.running := FALSE;
   c_mtrdir.status.old.fault := FALSE;
   c_mtrlin.enable := FALSE;
   c_mtrlin.index := 0;
   c_mtrlin.cmd := FALSE;
   c_mtrlin.fup := FALSE;
   c_mtrlin.status.running := FALSE;
   c_mtrlin.status.inFault := FALSE;
   c_mtrlin.status.justStarted := FALSE;
   c_mtrlin.status.justStopped := FALSE;
   c_mtrlin.status.justHadFault := FALSE;
   c_mtrlin.status.justLostFault := FALSE;
   c_mtrlin.status.reference := 0.0;
   c_mtrlin.status.enabled := FALSE;
   c_mtrlin.status.old.running := FALSE;
   c_mtrlin.status.old.fault := FALSE;
END_DATA_BLOCK

DATA_BLOCK "AlarmGroup"   // DB1
// stored: InstanceOfName AFB_AlarmF, InstanceOfType FB
"AFB_AlarmF"
BEGIN
   M_TYPE_FAULT[0] := 0;
   M_TYPE_FAULT[1] := 3;
   M_TYPE_FAULT[2] := 0;
   M_TYPE_FAULT[3] := 5;
   M_TYPE_FAULT[4] := 3;
   M_TYPE_FAULT[5] := 0;
   M_TYPE_FAULT[6] := 2;
   M_TYPE_FAULT[7] := 0;
   M_TYPE_FAULT[8] := 1;
   M_TYPE_WARNING[0] := 3;
   M_TYPE_WARNING[1] := 0;
   M_TYPE_WARNING[2] := 1;
   nFault.Alarm[0..5] := 0;
   nFault.Alarm[6] := 1;
   nFault.Alarm[7..8] := 0;
   nFault.Ackn[0] := 0;
   nFault.Ackn[1] := 8;
   nFault.Ackn[2] := 0;
   nFault.Ackn[3] := 13;
   nFault.Ackn[4] := 21;
   nFault.Ackn[5] := 0;
   nFault.Ackn[6] := 16;
   nFault.Ackn[7] := 4;
   nFault.Ackn[8] := 8;
   nFault.Siren[0..5] := 0;
   nFault.Siren[6] := 1;
   nFault.Siren[7..8] := 0;
   nWarning.Alarm[0..2] := 0;
   nWarning.Ackn[0] := 4;
   nWarning.Ackn[1] := 0;
   nWarning.Ackn[2] := 1;
   nWarning.Siren[0..2] := 0;
END_DATA_BLOCK

